(* IEC 61131-3 sources: Bachelor-s-thesis-RoboDK-PLC-interface-via-OPC-UA/robodk-codesys-opcua-interface/codesys, 2 files *)

(* ---- GVL.st ---- *)
VAR_GLOBAL

  (* Commands from the visualization / GUI *)

  Trigger : BOOL := FALSE;        // Signal to start the selected program

  Stop : BOOL := FALSE;           // Signal to stop the running program

  Selected_Index : INT := 0;      // Index of the selected program (1..MAX)

  (* Information from Python over OPC UA / feedback from RoboDK *)

  Robot_Run : BOOL := FALSE;      // Status: RoboDK standard program is running

  IO_Run : BOOL := FALSE;         // Status: RoboDK program (Python/standard) is running

  Current_Program : STRING(50) := '';       // Name of the program currently running

  Comb_names : ARRAY[1..50] OF STRING(80);  // List of all available programs

  Nb_Programs : INT := 0;         // Number of programs in the station

  (* Industrial IO - commands PLC -> RoboDK *)

  IO_ : ARRAY[1..50] OF BOOL := [FALSE];    // Control IOs PLC -> RoboDK

  (* Physical start button *)

  Start_IO : BOOL := FALSE;       // Manual start signal for industrial programs

END_VAR

(* ---- PLC_PRG.st ---- *)
PROGRAM PLC_PRG

VAR

  RStart       : R_TRIG;

  RisingStop   : R_TRIG;

  i            : INT;

END_VAR

(* Rising edge detection of the physical start button *)

RStart(CLK := Start_IO);

(* Rising edge detection of the stop button *)

RisingStop(CLK := Stop);

(* ===== STOP ===== *)

IF RisingStop.Q THEN

  Stop := TRUE; (* Latch the stop command *)

END_IF

IF Stop THEN

  (* Immediately reset all IO commands *)

  FOR i := 1 TO 50 DO

    IO_[i] := FALSE;

  END_FOR;

END_IF

(* ===== START ===== *)

IF RStart.Q THEN

  IF (Selected_Index >= 1) AND (Selected_Index <= Nb_Programs) THEN

    (* Reset all IO commands *)

    FOR i := 1 TO 50 DO

      IO_[i] := FALSE;

    END_FOR;

    (* Activate the IO that matches the selected program *)

    IO_[Selected_Index] := TRUE;

  END_IF;

  (* Reset the physical start button *)

  Start_IO := FALSE;

END_IF
